(* IEC 61131-3 sources: SmartHomeNew/snapshots/project_clean_state_2026_04_16/workspace/dut_rebuild/socket_v2/extraction, 1 file *)

(* ---- FB_Socket_State_Extractor_DRAFT.st ---- *)
FUNCTION_BLOCK FB_Socket_State_Extractor_DRAFT
VAR_INPUT
    VI_Is_On : BOOL;
    VI_Safety_Blocked : BOOL;
END_VAR
VAR_OUTPUT
    VO_State : ST_Socket_State_V2;
END_VAR

VO_State.Is_On := VI_Is_On;
VO_State.Safety_Blocked := VI_Safety_Blocked;
END_FUNCTION_BLOCK
